TYPE ST_EFU_Inputs :
STRUCT
	bWarning 	: BOOL;
	bError 		: BOOL;
	bTripped 	: BOOL;
	bEnabled 	: BOOL;
	//InputCycleCounter : BYTE;
	fCurrent 	: REAL;
END_STRUCT
END_TYPE

(* stored: Version 1.1.0.1
   DUT ST_EFU_Inputs: Id {7370842a-66da-4f0c-981f-c349e0bf9a26} *)
